// SIMATIC S7-200 project (STEP 7-Micro/WIN), CPU 226 REL 02.01

ORGANIZATION_BLOCK MAIN:OB1
TITLE=PROGRAM COMMENTS
BEGIN
Network 1 // 2^0 digit
LDN    I0.0
A      I1.0
LD     I0.0
AN     I1.0
OLD
=      Q0.0
Network 2
LDN    I0.1
AN     I1.1
A      I0.0
A      I1.0
LDN    I0.1
A      I1.1
LD     I0.0
A      I1.0
NOT
ALD
OLD
LD     I0.1
AN     I1.1
LD     I0.0
A      I1.0
NOT
ALD
OLD
LD     I0.1
A      I1.1
A      I0.0
A      I1.0
OLD
=      Q0.1
Network 3
LDN    I0.1
A      I1.1
A      I0.0
A      I1.0
LD     I0.1
AN     I1.1
A      I0.0
A      I1.0
OLD
LD     I0.1
A      I1.1
A      I0.0
A      I1.0
OLD
LD     I0.1
A      I1.1
LD     I0.0
A      I1.0
NOT
ALD
OLD
=      M0.1
Network 4
LDN    I0.2
AN     I1.2
A      M0.1
LDN    I0.2
A      I1.2
AN     M0.1
OLD
LD     I0.2
AN     I1.2
AN     M0.1
OLD
LD     I0.2
A      I1.2
A      M0.1
OLD
=      Q0.2
Network 5
LDN    I0.2
A      I1.2
A      M0.1
LD     I0.2
AN     I1.2
A      M0.1
OLD
LD     I0.2
A      I1.2
A      M0.1
OLD
LD     I0.2
A      I1.2
AN     M0.1
OLD
=      Q0.3
END_ORGANIZATION_BLOCK
